FUNCTION_BLOCK FB_Hmi_Led EXTENDS FB_Hmi_Component
VAR
	_rLed: REFERENCE TO S_Hmi_Led;

	_blink: BOOL;
	_blinkTime: TIME;
	_Blinker: FB_Timer;
END_VAR

IF _blink THEN
	IF _Blinker.Done THEN
		_Blinker.Start(_blinkTime);
		_rLed.OnOff := NOT _rLed.OnOff;
	END_IF
END_IF

PROPERTY PUBLIC Blink : BOOL
SET
_blink := Blink;
_rLed.OnOff := FALSE;
END_SET
END_PROPERTY

PROPERTY PUBLIC BlinkTime : TIME
SET
BlinkTime := _blinkTime;
END_SET
END_PROPERTY

METHOD PUBLIC Initialize : BOOL
VAR_INPUT
	rLed: REFERENCE TO S_Hmi_Led;
END_VAR
IF __ISVALIDREF(rLed) THEN
	_rLed REF= rLed;
	_initialized := Initialize := TRUE;
END_IF
END_METHOD

PROPERTY PUBLIC OffColor : UINT
SET
_rLed.OffColor := OffColor;
END_SET
END_PROPERTY

PROPERTY PUBLIC OnColor : UINT
SET
_rLed.OnColor := OnColor;
END_SET
END_PROPERTY

PROPERTY PUBLIC OnOff : BOOL
SET
_rLed.OnOff := OnOff;
END_SET
END_PROPERTY

PROPERTY PUBLIC Visibility : BOOL
SET
_rLed.Visibility := Visibility;
END_SET
END_PROPERTY

END_FUNCTION_BLOCK

(* stored: Version 1.1.0.1, ProductVersion 3.1.4024.10
   POU FB_Hmi_Led: Id {629fea12-c436-4ed1-9312-b78a6f33c585}, SpecialFunc None
   Property Blink: Id {24256100-f185-4ab0-9bd9-6faa3bcaa067}
   Set Set: Id {e73eeed1-a2fc-4be7-920d-2ff398949c89}
   Property BlinkTime: Id {cd96fd92-f08c-4627-8d73-44bcf2dd44c7}
   Set Set: Id {20b97150-0a5c-48b2-8668-ed751543bb5d}
   Method Initialize: Id {1f17b9b0-7303-42ad-8ed9-7054ea71c975}
   Property OffColor: Id {4493657e-7507-403f-85e1-b1f270d9f0a6}
   Set Set: Id {298e6dad-e893-4663-a6a0-9d73e5fe510f}
   Property OnColor: Id {6751ab28-320c-449b-9461-494d5cabf93d}
   Set Set: Id {f6b81999-6efb-45ba-a7c4-2290a3abc8af}
   Property OnOff: Id {7c2e37f6-22b6-4019-a01a-20f898899411}
   Set Set: Id {7f2ea347-8b3c-4369-9309-65fe19aa3ca3}
   Property Visibility: Id {f1ca3213-c9b8-41cb-bd21-2770983b098c}
   Set Set: Id {8af37679-8928-40a4-9810-0c143709bd3c} *)
